FUNCTION_BLOCK FB_ExampleDevice
VAR_INPUT
END_VAR
VAR_OUTPUT
END_VAR
VAR
	MC_MoveAbsolute_0: MC_MoveAbsolute;
	fbBCTM: BeamClassTransitionManager;
	FB_ExampleDeviceSM_0: FB_ExampleDeviceSM;
	stDevice	:	ST_Device;
	MC_Power_0: MC_Power;
	MC_Stop_0	:	MC_Stop;
END_VAR

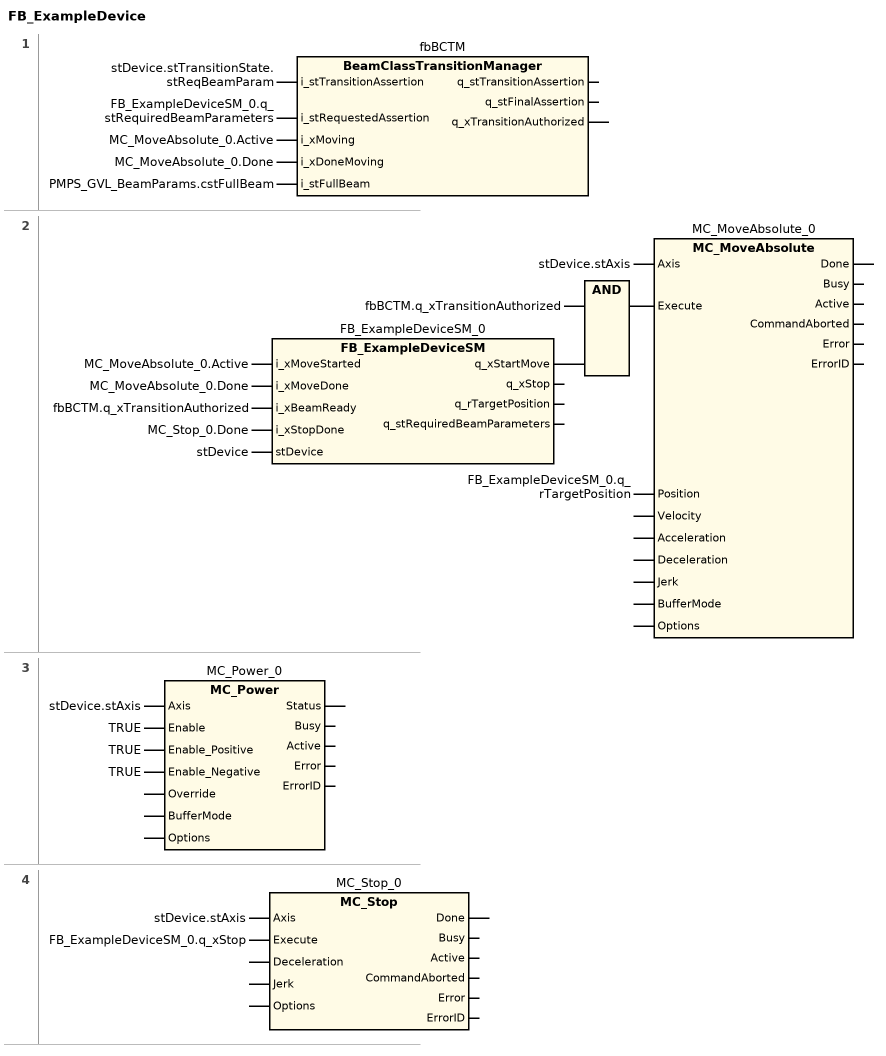
// NETWORK 1
fbBCTM(
    i_stTransitionAssertion := stDevice.stTransitionState.stReqBeamParam,
    i_stRequestedAssertion := FB_ExampleDeviceSM_0.q_stRequiredBeamParameters,
    i_xMoving := MC_MoveAbsolute_0.Active,
    i_xDoneMoving := MC_MoveAbsolute_0.Done,
    i_stFullBeam := PMPS_GVL_BeamParams.cstFullBeam); // BeamClassTransitionManager

// NETWORK 2
FB_ExampleDeviceSM_0(
    i_xMoveStarted := MC_MoveAbsolute_0.Active,
    i_xMoveDone := MC_MoveAbsolute_0.Done,
    i_xBeamReady := fbBCTM.q_xTransitionAuthorized,
    i_xStopDone := MC_Stop_0.Done,
    stDevice := stDevice); // FB_ExampleDeviceSM
MC_MoveAbsolute_0(
    Axis := stDevice.stAxis,
    Execute := fbBCTM.q_xTransitionAuthorized AND FB_ExampleDeviceSM_0.q_xStartMove,
    Position := FB_ExampleDeviceSM_0.q_rTargetPosition); // MC_MoveAbsolute

// NETWORK 3
MC_Power_0(Axis := stDevice.stAxis, Enable := TRUE, Enable_Positive := TRUE, Enable_Negative := TRUE); // MC_Power

// NETWORK 4
MC_Stop_0(Axis := stDevice.stAxis, Execute := FB_ExampleDeviceSM_0.q_xStop); // MC_Stop

ACTION Initialize:

stDevice.astStates[1].rPosition := 100;
stDevice.astStates[1].nStateRef := 16#1;
stDevice.astStates[1].stReqBeamParam := F_SetBeamParams(
	fAtt := 20,
	fPP_mJ := 1,
	fLower_eV := 0,
	fUpper_eV := 1500
);

stDevice.astStates[2].rPosition := 200;
stDevice.astStates[1].nStateRef := 16#2;
stDevice.astStates[2].stReqBeamParam := F_SetBeamParams(
	fAtt := 50,
	fPP_mJ := 1,
	fLower_eV := 0,
	fUpper_eV := 1500
);

stDevice.astStates[3].rPosition := 300;
stDevice.astStates[1].nStateRef := 16#3;
stDevice.astStates[3].stReqBeamParam := F_SetBeamParams(
	fAtt := 50,
	fPP_mJ := 0.5,
	fLower_eV := 0,
	fUpper_eV := 1500
);

stDevice.stTransitionState.nStateRef := 16#10;
stDevice.stTransitionState.stReqBeamParam := F_SetBeamParams(
	fAtt := 100,
	fPP_mJ := 1,
	fLower_eV := 0,
	fUpper_eV := 1500
);
END_ACTION

END_FUNCTION_BLOCK

(* stored: Version 1.1.0.1, ProductVersion 3.1.4022.12
   POU FB_ExampleDevice: Id {1f4ba9e5-9568-049e-05f4-859598559522}, SpecialFunc None
   Action Initialize: Id {00e2bf73-95c1-07cf-3db2-5bb9d2dbc900} *)
